PROGRAM AUTO_SCREWLENGTH
VAR
END_VAR

END_PROGRAM

(* stored: Version 1.1.0.1, ProductVersion 3.1.4022.18
   POU AUTO_SCREWLENGTH: Id {0204b2d1-fbb4-4780-b187-5cd2aeb8d721}, SpecialFunc None *)
